{attribute addProperty BoxType "EL2564-0000-0016"}
{attribute addProperty Id "PWM_Inputs_ChannelAT %I*ARRAY[0..3] OF PWM_Inputs_Channel_35DD72E46480PWM_Outputs_ChannelAT %Q*ARRAY[0..3] OF PWM_Outputs_Channel_FAB5DC8C6480WcStateAT %I*WcState_98A4DF7520.250InfoDataAT %I*InfoData_BC63D37F80100"}
{attribute addProperty CRC "807394020"}
{attribute addProperty SizeInBites "210"}
{attribute addProperty SizeInBytes "26.25"}
TYPE EL2564_D618E7A6 :
STRUCT
	{attribute addProperty Name "PWM_Inputs_Channel"}
	PWM_Inputs_Channel : ARRAY[0..3] OF PWM_Inputs_Channel_35DD72E4;
	{attribute addProperty Name "PWM_Outputs_Channel"}
	PWM_Outputs_Channel : ARRAY[0..3] OF PWM_Outputs_Channel_FAB5DC8C;
	{attribute addProperty Name "WcState"}
	WcState : WcState_98A4DF75;
	{attribute addProperty Name "InfoData"}
	InfoData : InfoData_BC63D37F;
END_STRUCT
END_TYPE

(* stored: Version 1.2.0.0, ProductVersion 3.1.4024.9
   DUT EL2564_D618E7A6: Id {9c3d6dd3-a256-40d4-a8c0-5687378333c4} *)
